(* Schneider Machine Expert - Basic project 3 Pompes permutation temporelle, file version 2.8.0.0 *)
(* ProjectInformations: Name=New project *)

HARDWARE
  Cpu 0: TM221CE40T
  ModuleExtensionObject 0: TM3AI2H/G
  EthernetConfiguration: NetworkName=M221, IpAllocationMode=FixedAddress, IpAddress=192.168.1.11, SubnetMask=255.255.255.0
  SerialLineConfiguration: Baud=Baud19200, Parity=ParityEven, DataBits=DataBits8, StopBits=StopBits1, PhysicalMedium=PhysicalMediumRs485, TransmissionMode=TransmissionModeModbusRtu, SlaveId=1, Addressing=SlaveAddressing
  MastTask: UsePeriodScanMode=false, PeriodScan=100
  FastTask: Period=255
  CpuBehavior: StartingMode=StartAsPreviousState, AutoSaveRamOnEeprom=true, WatchdogPeriod=250

SYMBOLS  (address, symbol, comment, settings)
  %M0       SEL_POMPE
  %M1       RESET_SELECTEUR
  %M5       MODE_1P
  %M6       MODE_2P
  %S6       SB_TB1S  "Time base of 1 s generated by an internal clock"
  %MW0      CHOIX_POMPE
  %MD10     TEMPS_P1
  %MD12     TEMPS_P2
  %MD14     TEMPS_P3
  %C0       SELECTEUR  [Preset=2]
  %I0.0     BP_MARCHE
  %I0.1     BP_ARRET
  %I0.2     SURCHAUFFE_1
  %I0.3     RESET
  %I0.4     POIRE_NTB
  %I0.5     ARR_URG
  %I0.6     SURCHAUFFE_2
  %I0.7     SURCHAUFFE_3
  %Q0.0     MARCHE_P1
  %Q0.1     V_MARCHE_1
  %Q0.2     V_ARRET_1
  %Q0.3     V_DEFAUT_1
  %Q0.4     MARCHE_P2
  %Q0.5     V_MARCHE_2
  %Q0.6     V_ARRET_2
  %Q0.7     V_DEFAUT_2
  %Q0.8     V_MARCHE_3
  %Q0.9     V_ARRET_3
  %Q0.10    V_DEFAUT_3
  %Q0.11    MARCHE_P3
  %IW1.0    NIV_RES  [Type=Type_4_20mA, Scope=Scope_Customized, Minimum=0, Maximum=500]

POU Protection
  (* SectionNumber=1 *)

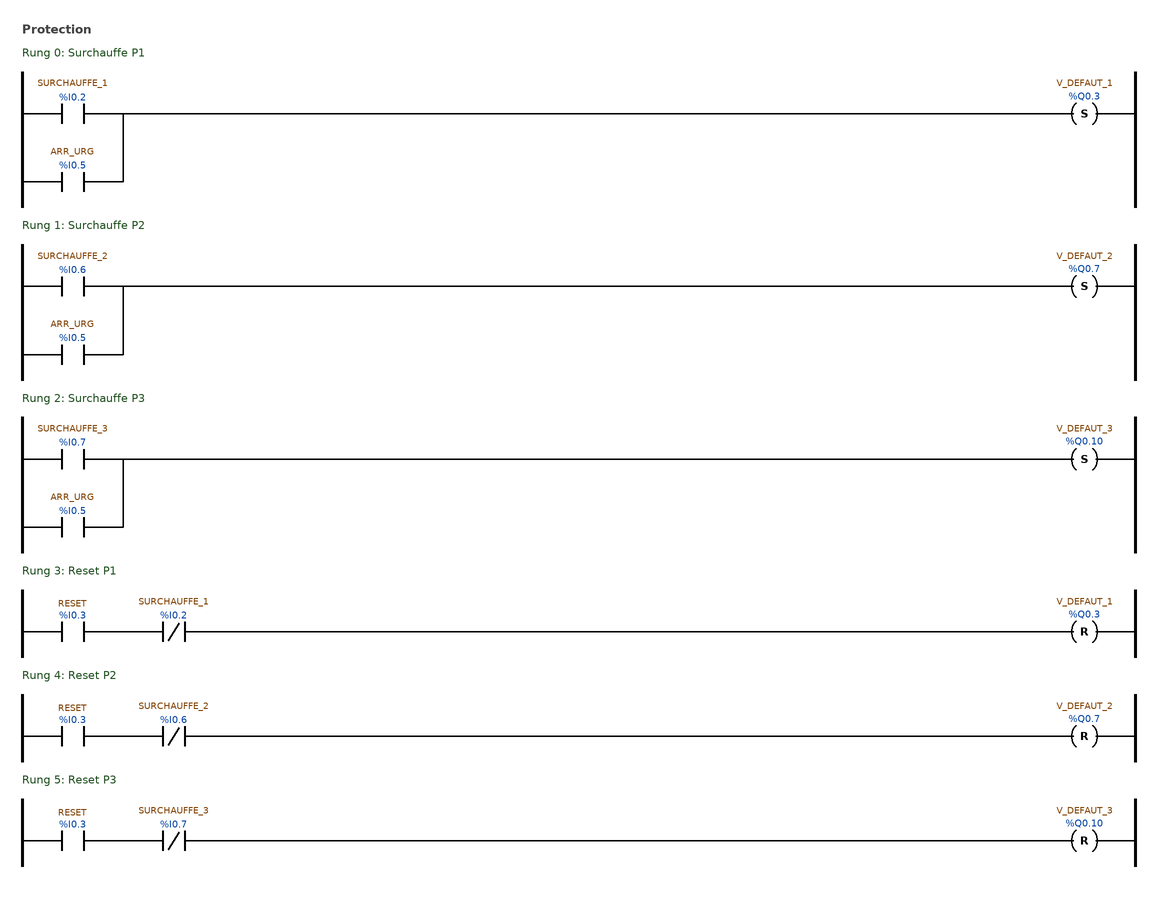

// Rung 0: Surchauffe P1
  LD %I0.2                (* SURCHAUFFE_1 *)
  OR %I0.5                (* ARR_URG *)
  S %Q0.3                 (* V_DEFAUT_1 *)
  // as ST:
  //   IF SURCHAUFFE_1 OR ARR_URG THEN V_DEFAUT_1 := TRUE; END_IF;

// Rung 1: Surchauffe P2
  LD %I0.6                (* SURCHAUFFE_2 *)
  OR %I0.5                (* ARR_URG *)
  S %Q0.7                 (* V_DEFAUT_2 *)
  // as ST:
  //   IF SURCHAUFFE_2 OR ARR_URG THEN V_DEFAUT_2 := TRUE; END_IF;

// Rung 2: Surchauffe P3
  LD %I0.7                (* SURCHAUFFE_3 *)
  OR %I0.5                (* ARR_URG *)
  S %Q0.10                (* V_DEFAUT_3 *)
  // as ST:
  //   IF SURCHAUFFE_3 OR ARR_URG THEN V_DEFAUT_3 := TRUE; END_IF;

// Rung 3: Reset P1
  LD %I0.3                (* RESET *)
  ANDN %I0.2              (* SURCHAUFFE_1 *)
  R %Q0.3                 (* V_DEFAUT_1 *)
  // as ST:
  //   IF RESET AND NOT SURCHAUFFE_1 THEN V_DEFAUT_1 := FALSE; END_IF;

// Rung 4: Reset P2
  LD %I0.3                (* RESET *)
  ANDN %I0.6              (* SURCHAUFFE_2 *)
  R %Q0.7                 (* V_DEFAUT_2 *)
  // as ST:
  //   IF RESET AND NOT SURCHAUFFE_2 THEN V_DEFAUT_2 := FALSE; END_IF;

// Rung 5: Reset P3
  LD %I0.3                (* RESET *)
  ANDN %I0.7              (* SURCHAUFFE_3 *)
  R %Q0.10                (* V_DEFAUT_3 *)
  // as ST:
  //   IF RESET AND NOT SURCHAUFFE_3 THEN V_DEFAUT_3 := FALSE; END_IF;

POU Marche P1
  (* SectionNumber=2 *)

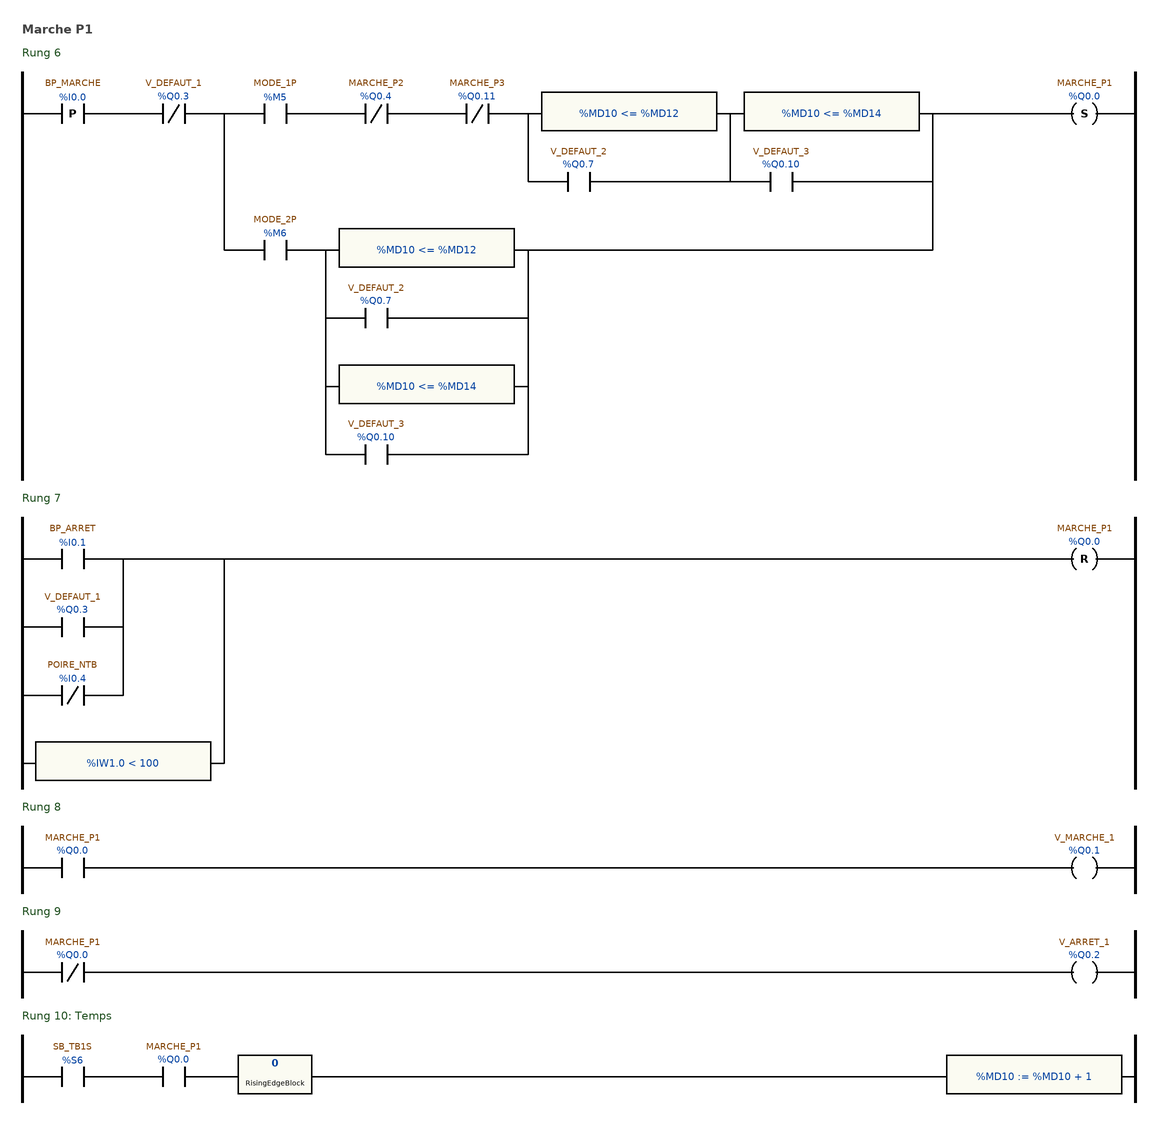

// Rung 6
  LDR %I0.0               (* BP_MARCHE *)
  ANDN %Q0.3              (* V_DEFAUT_1 *)
  AND( %M5                (* MODE_1P *)
  ANDN %Q0.4              (* MARCHE_P2 *)
  ANDN %Q0.11             (* MARCHE_P3 *)
  AND( [ %MD10 <= %MD12 ] (* TEMPS_P1, TEMPS_P2 *)
  OR %Q0.7                (* V_DEFAUT_2 *)
  )
  AND( [ %MD10 <= %MD14 ] (* TEMPS_P1, TEMPS_P3 *)
  OR %Q0.10               (* V_DEFAUT_3 *)
  )
  OR( %M6                 (* MODE_2P *)
  AND( [ %MD10 <= %MD12 ] (* TEMPS_P1, TEMPS_P2 *)
  OR %Q0.7                (* V_DEFAUT_2 *)
  OR [ %MD10 <= %MD14 ]   (* TEMPS_P1, TEMPS_P3 *)
  OR %Q0.10               (* V_DEFAUT_3 *)
  )
  )
  )
  S %Q0.0                 (* MARCHE_P1 *)
  // as ST:
  //   IF RISING(BP_MARCHE) AND NOT V_DEFAUT_1 AND (MODE_1P AND NOT MARCHE_P2 AND NOT MARCHE_P3 AND (TEMPS_P1 <= TEMPS_P2 OR V_DEFAUT_2) AND (TEMPS_P1 <= TEMPS_P3 OR V_DEFAUT_3) OR MODE_2P AND (TEMPS_P1 <= TEMPS_P2 OR V_DEFAUT_2 OR TEMPS_P1 <= TEMPS_P3 OR V_DEFAUT_3)) THEN MARCHE_P1 := TRUE; END_IF;

// Rung 7
  LD %I0.1                (* BP_ARRET *)
  OR %Q0.3                (* V_DEFAUT_1 *)
  ORN %I0.4               (* POIRE_NTB *)
  OR [ %IW1.0 < 100 ]     (* NIV_RES *)
  R %Q0.0                 (* MARCHE_P1 *)
  // as ST:
  //   IF BP_ARRET OR V_DEFAUT_1 OR NOT POIRE_NTB OR NIV_RES < 100 THEN MARCHE_P1 := FALSE; END_IF;

// Rung 8
  LD %Q0.0                (* MARCHE_P1 *)
  ST %Q0.1                (* V_MARCHE_1 *)
  // as ST:
  //   V_MARCHE_1 := MARCHE_P1;

// Rung 9
  LDN %Q0.0               (* MARCHE_P1 *)
  ST %Q0.2                (* V_ARRET_1 *)
  // as ST:
  //   V_ARRET_1 := NOT MARCHE_P1;

// Rung 10: Temps
  LD %S6                  (* SB_TB1S *)
  AND %Q0.0               (* MARCHE_P1 *)
  RISING0
  [ %MD10 := %MD10 + 1 ]  (* TEMPS_P1, TEMPS_P1 *)
  // as ST:
  //   IF RISING(SB_TB1S AND MARCHE_P1) THEN TEMPS_P1 := TEMPS_P1 + 1; END_IF;

POU Marche P2
  (* SectionNumber=3 *)

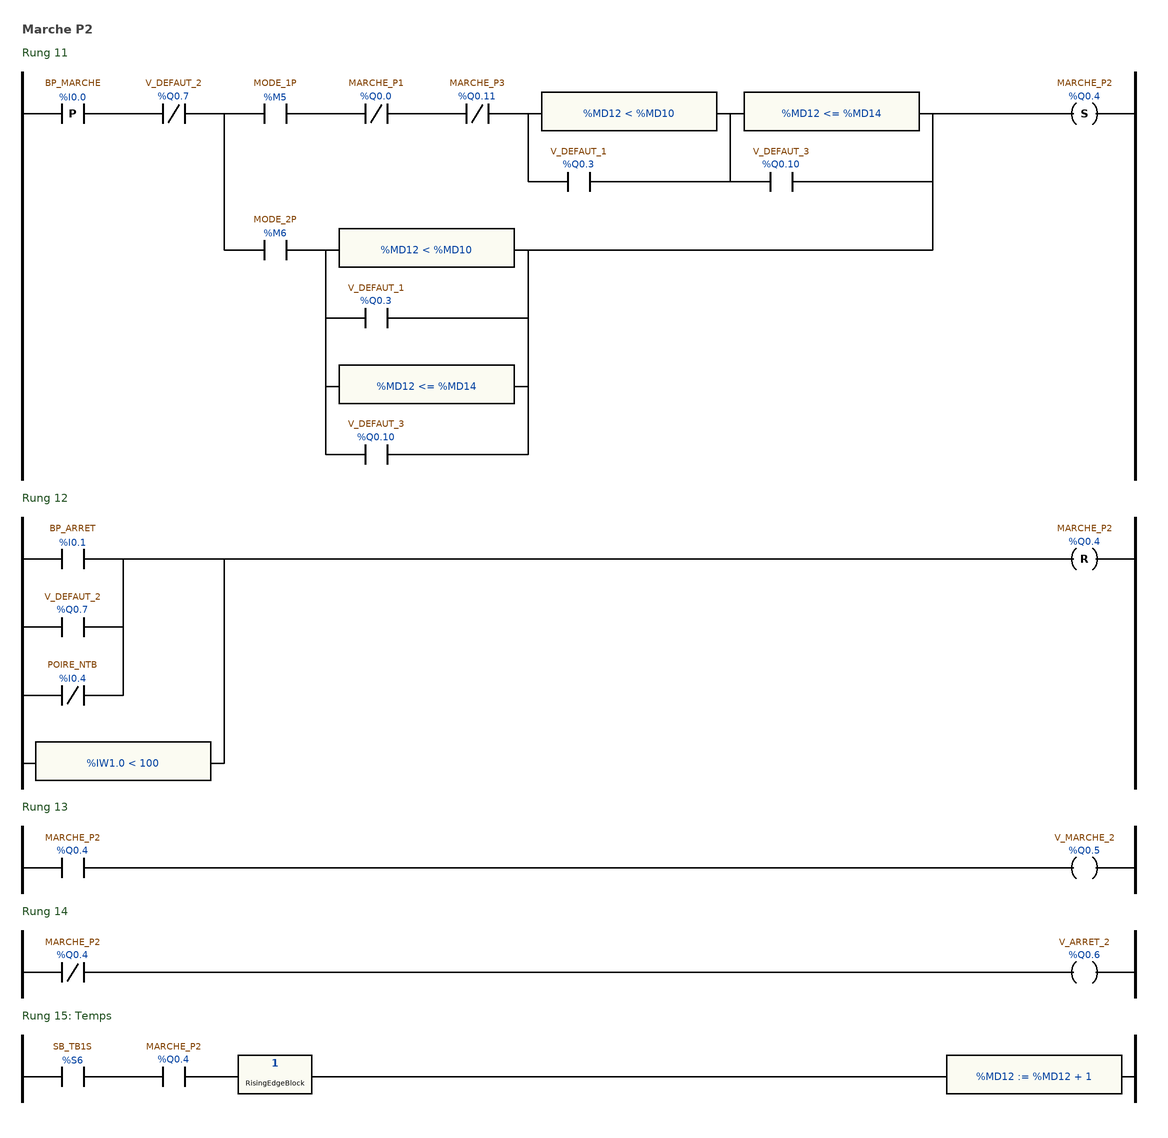

// Rung 11
  LDR %I0.0               (* BP_MARCHE *)
  ANDN %Q0.7              (* V_DEFAUT_2 *)
  AND( %M5                (* MODE_1P *)
  ANDN %Q0.0              (* MARCHE_P1 *)
  ANDN %Q0.11             (* MARCHE_P3 *)
  AND( [ %MD12 < %MD10 ]  (* TEMPS_P2, TEMPS_P1 *)
  OR %Q0.3                (* V_DEFAUT_1 *)
  )
  AND( [ %MD12 <= %MD14 ] (* TEMPS_P2, TEMPS_P3 *)
  OR %Q0.10               (* V_DEFAUT_3 *)
  )
  OR( %M6                 (* MODE_2P *)
  AND( [ %MD12 < %MD10 ]  (* TEMPS_P2, TEMPS_P1 *)
  OR %Q0.3                (* V_DEFAUT_1 *)
  OR [ %MD12 <= %MD14 ]   (* TEMPS_P2, TEMPS_P3 *)
  OR %Q0.10               (* V_DEFAUT_3 *)
  )
  )
  )
  S %Q0.4                 (* MARCHE_P2 *)
  // as ST:
  //   IF RISING(BP_MARCHE) AND NOT V_DEFAUT_2 AND (MODE_1P AND NOT MARCHE_P1 AND NOT MARCHE_P3 AND (TEMPS_P2 < TEMPS_P1 OR V_DEFAUT_1) AND (TEMPS_P2 <= TEMPS_P3 OR V_DEFAUT_3) OR MODE_2P AND (TEMPS_P2 < TEMPS_P1 OR V_DEFAUT_1 OR TEMPS_P2 <= TEMPS_P3 OR V_DEFAUT_3)) THEN MARCHE_P2 := TRUE; END_IF;

// Rung 12
  LD %I0.1                (* BP_ARRET *)
  OR %Q0.7                (* V_DEFAUT_2 *)
  ORN %I0.4               (* POIRE_NTB *)
  OR [ %IW1.0 < 100 ]     (* NIV_RES *)
  R %Q0.4                 (* MARCHE_P2 *)
  // as ST:
  //   IF BP_ARRET OR V_DEFAUT_2 OR NOT POIRE_NTB OR NIV_RES < 100 THEN MARCHE_P2 := FALSE; END_IF;

// Rung 13
  LD %Q0.4                (* MARCHE_P2 *)
  ST %Q0.5                (* V_MARCHE_2 *)
  // as ST:
  //   V_MARCHE_2 := MARCHE_P2;

// Rung 14
  LDN %Q0.4               (* MARCHE_P2 *)
  ST %Q0.6                (* V_ARRET_2 *)
  // as ST:
  //   V_ARRET_2 := NOT MARCHE_P2;

// Rung 15: Temps
  LD %S6                  (* SB_TB1S *)
  AND %Q0.4               (* MARCHE_P2 *)
  RISING1
  [ %MD12 := %MD12 + 1 ]  (* TEMPS_P2, TEMPS_P2 *)
  // as ST:
  //   IF RISING(SB_TB1S AND MARCHE_P2) THEN TEMPS_P2 := TEMPS_P2 + 1; END_IF;

POU Marche P3
  (* SectionNumber=4 *)

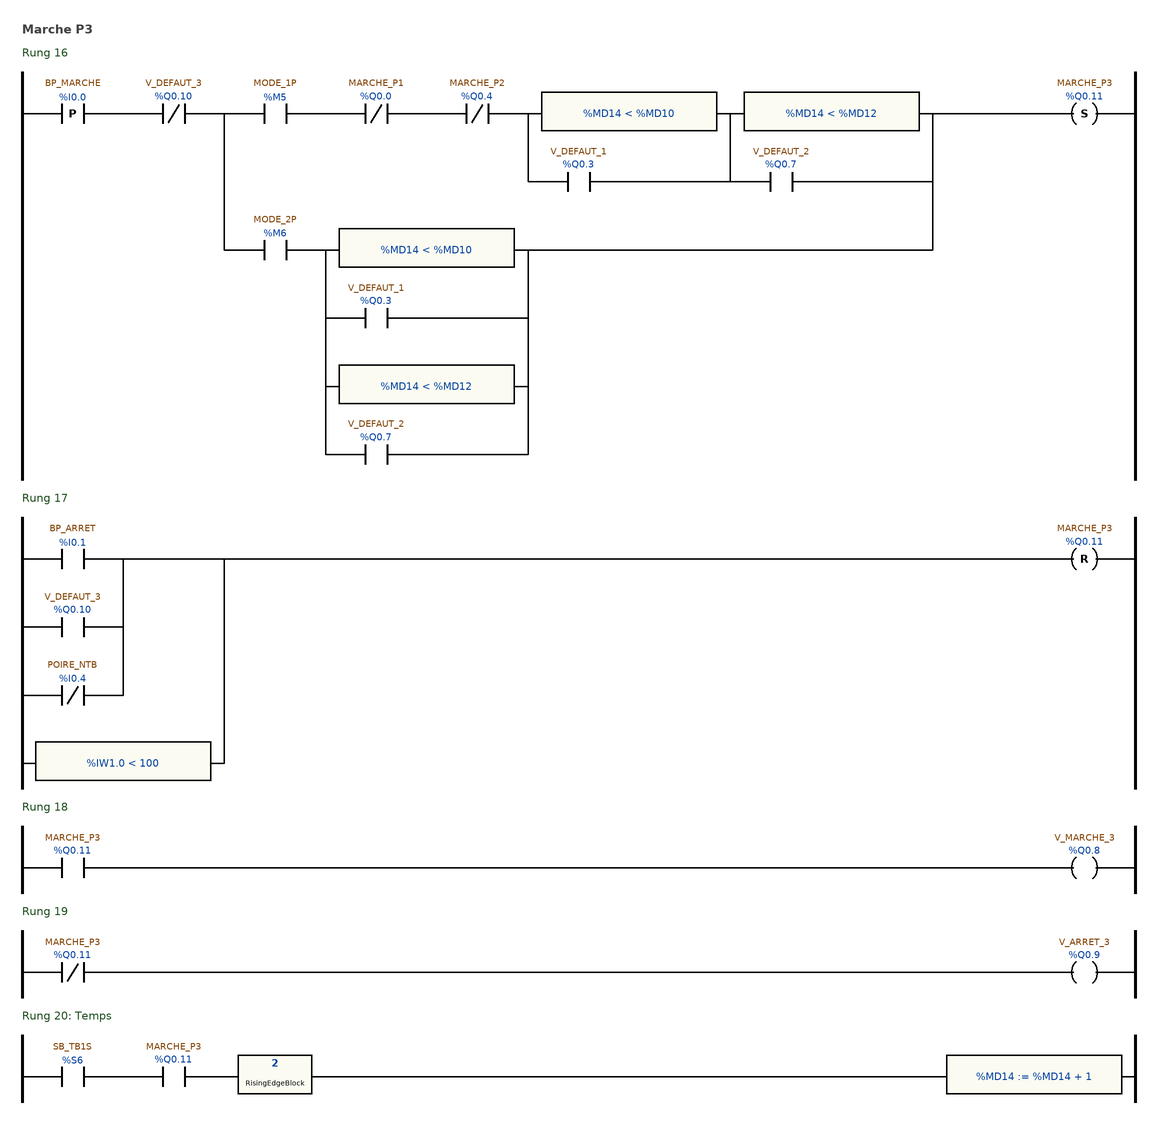

// Rung 16
  LDR %I0.0               (* BP_MARCHE *)
  ANDN %Q0.10             (* V_DEFAUT_3 *)
  AND( %M5                (* MODE_1P *)
  ANDN %Q0.0              (* MARCHE_P1 *)
  ANDN %Q0.4              (* MARCHE_P2 *)
  AND( [ %MD14 < %MD10 ]  (* TEMPS_P3, TEMPS_P1 *)
  OR %Q0.3                (* V_DEFAUT_1 *)
  )
  AND( [ %MD14 < %MD12 ]  (* TEMPS_P3, TEMPS_P2 *)
  OR %Q0.7                (* V_DEFAUT_2 *)
  )
  OR( %M6                 (* MODE_2P *)
  AND( [ %MD14 < %MD10 ]  (* TEMPS_P3, TEMPS_P1 *)
  OR %Q0.3                (* V_DEFAUT_1 *)
  OR [ %MD14 < %MD12 ]    (* TEMPS_P3, TEMPS_P2 *)
  OR %Q0.7                (* V_DEFAUT_2 *)
  )
  )
  )
  S %Q0.11                (* MARCHE_P3 *)
  // as ST:
  //   IF RISING(BP_MARCHE) AND NOT V_DEFAUT_3 AND (MODE_1P AND NOT MARCHE_P1 AND NOT MARCHE_P2 AND (TEMPS_P3 < TEMPS_P1 OR V_DEFAUT_1) AND (TEMPS_P3 < TEMPS_P2 OR V_DEFAUT_2) OR MODE_2P AND (TEMPS_P3 < TEMPS_P1 OR V_DEFAUT_1 OR TEMPS_P3 < TEMPS_P2 OR V_DEFAUT_2)) THEN MARCHE_P3 := TRUE; END_IF;

// Rung 17
  LD %I0.1                (* BP_ARRET *)
  OR %Q0.10               (* V_DEFAUT_3 *)
  ORN %I0.4               (* POIRE_NTB *)
  OR [ %IW1.0 < 100 ]     (* NIV_RES *)
  R %Q0.11                (* MARCHE_P3 *)
  // as ST:
  //   IF BP_ARRET OR V_DEFAUT_3 OR NOT POIRE_NTB OR NIV_RES < 100 THEN MARCHE_P3 := FALSE; END_IF;

// Rung 18
  LD %Q0.11               (* MARCHE_P3 *)
  ST %Q0.8                (* V_MARCHE_3 *)
  // as ST:
  //   V_MARCHE_3 := MARCHE_P3;

// Rung 19
  LDN %Q0.11              (* MARCHE_P3 *)
  ST %Q0.9                (* V_ARRET_3 *)
  // as ST:
  //   V_ARRET_3 := NOT MARCHE_P3;

// Rung 20: Temps
  LD %S6                  (* SB_TB1S *)
  AND %Q0.11              (* MARCHE_P3 *)
  RISING2
  [ %MD14 := %MD14 + 1 ]  (* TEMPS_P3, TEMPS_P3 *)
  // as ST:
  //   IF RISING(SB_TB1S AND MARCHE_P3) THEN TEMPS_P3 := TEMPS_P3 + 1; END_IF;

POU Mode 1P
  (* SectionNumber=5 *)

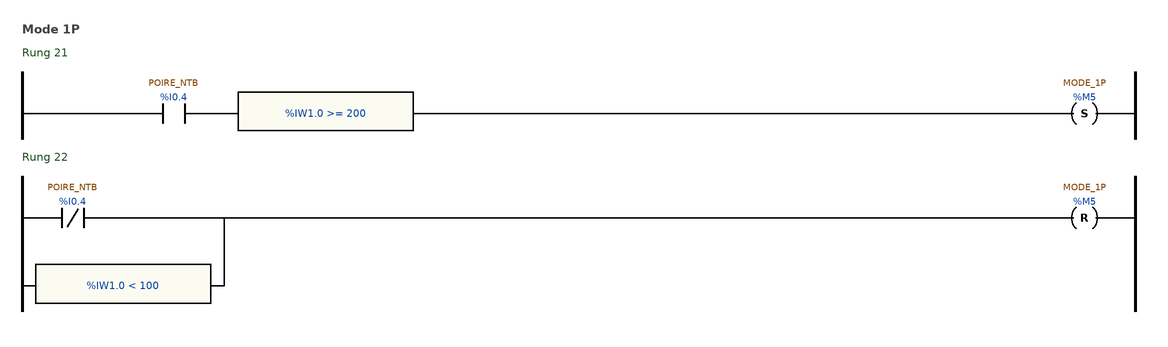

// Rung 21
  LD %I0.4                (* POIRE_NTB *)
  AND [ %IW1.0 >= 200 ]   (* NIV_RES *)
  S %M5                   (* MODE_1P *)
  // as ST:
  //   IF POIRE_NTB AND NIV_RES >= 200 THEN MODE_1P := TRUE; END_IF;

// Rung 22
  LDN %I0.4               (* POIRE_NTB *)
  OR [ %IW1.0 < 100 ]     (* NIV_RES *)
  R %M5                   (* MODE_1P *)
  // as ST:
  //   IF NOT POIRE_NTB OR NIV_RES < 100 THEN MODE_1P := FALSE; END_IF;

POU Mode 2P
  (* SectionNumber=6 *)

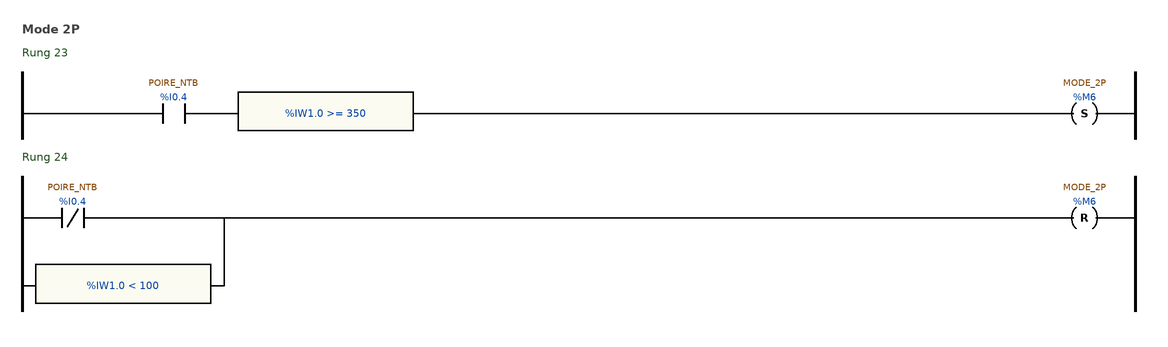

// Rung 23
  LD %I0.4                (* POIRE_NTB *)
  AND [ %IW1.0 >= 350 ]   (* NIV_RES *)
  S %M6                   (* MODE_2P *)
  // as ST:
  //   IF POIRE_NTB AND NIV_RES >= 350 THEN MODE_2P := TRUE; END_IF;

// Rung 24
  LDN %I0.4               (* POIRE_NTB *)
  OR [ %IW1.0 < 100 ]     (* NIV_RES *)
  R %M6                   (* MODE_2P *)
  // as ST:
  //   IF NOT POIRE_NTB OR NIV_RES < 100 THEN MODE_2P := FALSE; END_IF;
